FUNCTION_BLOCK FB_Motors
VAR_INPUT
	inIntlkOK : BOOL;
	inStart : BOOL;
END_VAR
VAR_OUTPUT
	outOTE: BOOL;
	outRunning : bool;
	outStopped : BOOL;
END_VAR
VAR
END_VAR

IF inIntlkOK AND inStart THEN
	outOTE := TRUE;
	outRunning := TRUE;
	outStopped := FALSE;
	ELSE
	outStopped := TRUE;
	outRunning := FALSE;
	outOTE := FALSE;
END_IF

END_FUNCTION_BLOCK

(* stored: Version 1.1.0.1
   POU FB_Motors: Id {1ee8bdc1-132c-42da-97d8-464190c90e99}, SpecialFunc None *)
